// SIMATIC S7-200 project (STEP 7-Micro/WIN), CPU 224XP REL 02.01

SYMBOL_TABLE USUARIO1
P_PEATONES       I0.0
C_ROJO           Q0.0
C_AMBAR          Q0.1
C_VERDE          Q0.2
P_ROJO           Q0.3
P_VERDE          Q0.4
AUXILIAR         Q2.0
SEGURIDAD        Q2.1
M_INTERMITENCIA  Q2.2
M2_INTERMITENCIA Q2.3
REINICIO_COCHES  Q3.1
REINICIO_PEATONES Q3.0
END_SYMBOL_TABLE

ORGANIZATION_BLOCK PRINCIPAL:OB1
TITLE=COMENTARIOS DEL PROGRAMA
BEGIN
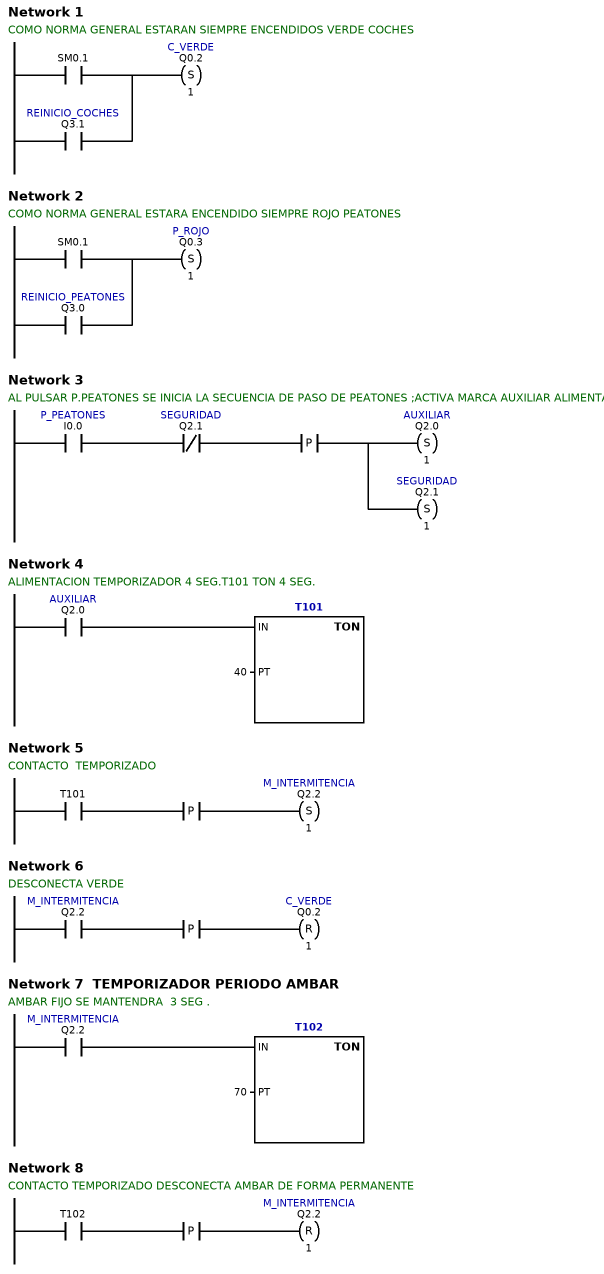
Network 1
// COMO NORMA GENERAL ESTARAN SIEMPRE ENCENDIDOS VERDE COCHES 
LD     SM0.1
O      REINICIO_COCHES:Q3.1
S      C_VERDE:Q0.2, 1
Network 2
// COMO NORMA GENERAL ESTARA ENCENDIDO SIEMPRE ROJO PEATONES
LD     SM0.1
O      REINICIO_PEATONES:Q3.0
S      P_ROJO:Q0.3, 1
Network 3
// AL PULSAR P.PEATONES SE INICIA LA SECUENCIA DE PASO DE PEATONES ;ACTIVA MARCA AUXILIAR ALIMENTACION Y MARCA SEGURIDAD PARA EVITAR EL INICIO UNA VEZ HALLA COMENZADO
LD     P_PEATONES:I0.0
AN     SEGURIDAD:Q2.1
EU
S      AUXILIAR:Q2.0, 1
S      SEGURIDAD:Q2.1, 1
Network 4
// ALIMENTACION TEMPORIZADOR 4 SEG.T101 TON 4 SEG.
LD     AUXILIAR:Q2.0
TON    T101, 40
Network 5
// CONTACTO  TEMPORIZADO 
LD     T101
EU
S      M_INTERMITENCIA:Q2.2, 1
Network 6
// DESCONECTA VERDE
LD     M_INTERMITENCIA:Q2.2
EU
R      C_VERDE:Q0.2, 1
Network 7 // TEMPORIZADOR PERIODO AMBAR
// AMBAR FIJO SE MANTENDRA  3 SEG . 
LD     M_INTERMITENCIA:Q2.2
TON    T102, 70
Network 8
// CONTACTO TEMPORIZADO DESCONECTA AMBAR DE FORMA PERMANENTE
LD     T102
EU
R      M_INTERMITENCIA:Q2.2, 1
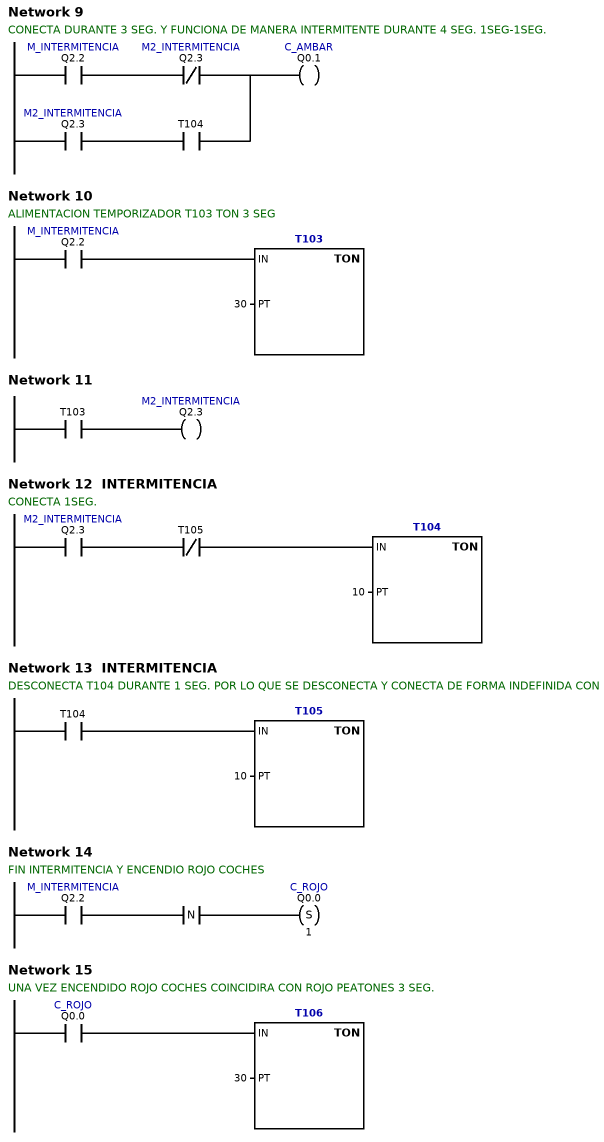
Network 9
// CONECTA DURANTE 3 SEG. Y FUNCIONA DE MANERA INTERMITENTE DURANTE 4 SEG. 1SEG-1SEG.
LD     M_INTERMITENCIA:Q2.2
AN     M2_INTERMITENCIA:Q2.3
LD     M2_INTERMITENCIA:Q2.3
A      T104
OLD
=      C_AMBAR:Q0.1
Network 10
// ALIMENTACION TEMPORIZADOR T103 TON 3 SEG
LD     M_INTERMITENCIA:Q2.2
TON    T103, 30
Network 11
LD     T103
=      M2_INTERMITENCIA:Q2.3
Network 12 // INTERMITENCIA
// CONECTA 1SEG.
LD     M2_INTERMITENCIA:Q2.3
AN     T105
TON    T104, 10
Network 13 // INTERMITENCIA
// DESCONECTA T104 DURANTE 1 SEG. POR LO QUE SE DESCONECTA Y CONECTA DE FORMA INDEFINIDA CON INTERVAL0 1SEG-1SEG.
LD     T104
TON    T105, 10
Network 14
// FIN INTERMITENCIA Y ENCENDIO ROJO COCHES 
LD     M_INTERMITENCIA:Q2.2
ED
S      C_ROJO:Q0.0, 1
Network 15
// UNA VEZ ENCENDIDO ROJO COCHES COINCIDIRA CON ROJO PEATONES 3 SEG.
LD     C_ROJO:Q0.0
TON    T106, 30
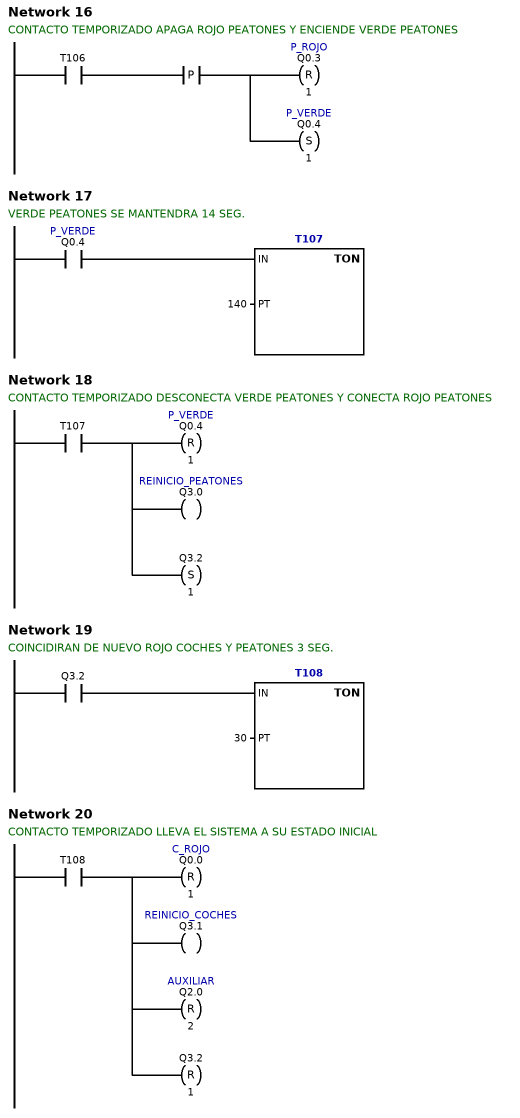
Network 16
// CONTACTO TEMPORIZADO APAGA ROJO PEATONES Y ENCIENDE VERDE PEATONES
LD     T106
EU
R      P_ROJO:Q0.3, 1
S      P_VERDE:Q0.4, 1
Network 17
// VERDE PEATONES SE MANTENDRA 14 SEG.
LD     P_VERDE:Q0.4
TON    T107, 140
Network 18
// CONTACTO TEMPORIZADO DESCONECTA VERDE PEATONES Y CONECTA ROJO PEATONES 
LD     T107
R      P_VERDE:Q0.4, 1
=      REINICIO_PEATONES:Q3.0
S      Q3.2, 1
Network 19
// COINCIDIRAN DE NUEVO ROJO COCHES Y PEATONES 3 SEG.
LD     Q3.2
TON    T108, 30
Network 20
// CONTACTO TEMPORIZADO LLEVA EL SISTEMA A SU ESTADO INICIAL
LD     T108
R      C_ROJO:Q0.0, 1
=      REINICIO_COCHES:Q3.1
R      AUXILIAR:Q2.0, 2
R      Q3.2, 1
END_ORGANIZATION_BLOCK
